// TIA Portal V17 export
// export: Created 2025-06-26T06:49:17.7875276Z, ExportSetting WithDefaults, DisplayName Totally Integrated Automation Portal, DisplayVersion V17 Update 8, DisplayName TIA Portal Openness, DisplayVersion V17 Update 8, DisplayName TIA Portal Version Control Interface, DisplayVersion V17, DisplayName STEP 7 Professional, DisplayVersion V17 Update 8, DisplayName STEP 7 Safety, DisplayVersion V17 Update 6, DisplayName WinCC Advanced, DisplayVersion V17 Update 8
FUNCTION "CompressorCalculations" : Void   // FC25, FBD
{ S7_Optimized_Access := 'TRUE' }
VERSION : 0.1
// stored: AutoNumber true, IsIECCheckEnabled false, SetENOAutomatically false, UDAEnableTagReadback false
   VAR_TEMP
      CrankcaseSaturationTemperature : Real;
      SaturationTemperatureSuction : Real;
      SaturationTemperatureDischarge : Real;
      Massflow : Real;
      VolumetricEfficiency : Real;
      HeatRateCompressor : Real;
      IsentropicEfficiencyCompressor : Real;
      FMEP : Real;
   END_VAR
   VAR_TEMP   // added for the SCL form of the ladder/FBD networks
      _w1 : Bool;
   END_VAR
BEGIN

REGION Network 1: Crankcase saturation temperature
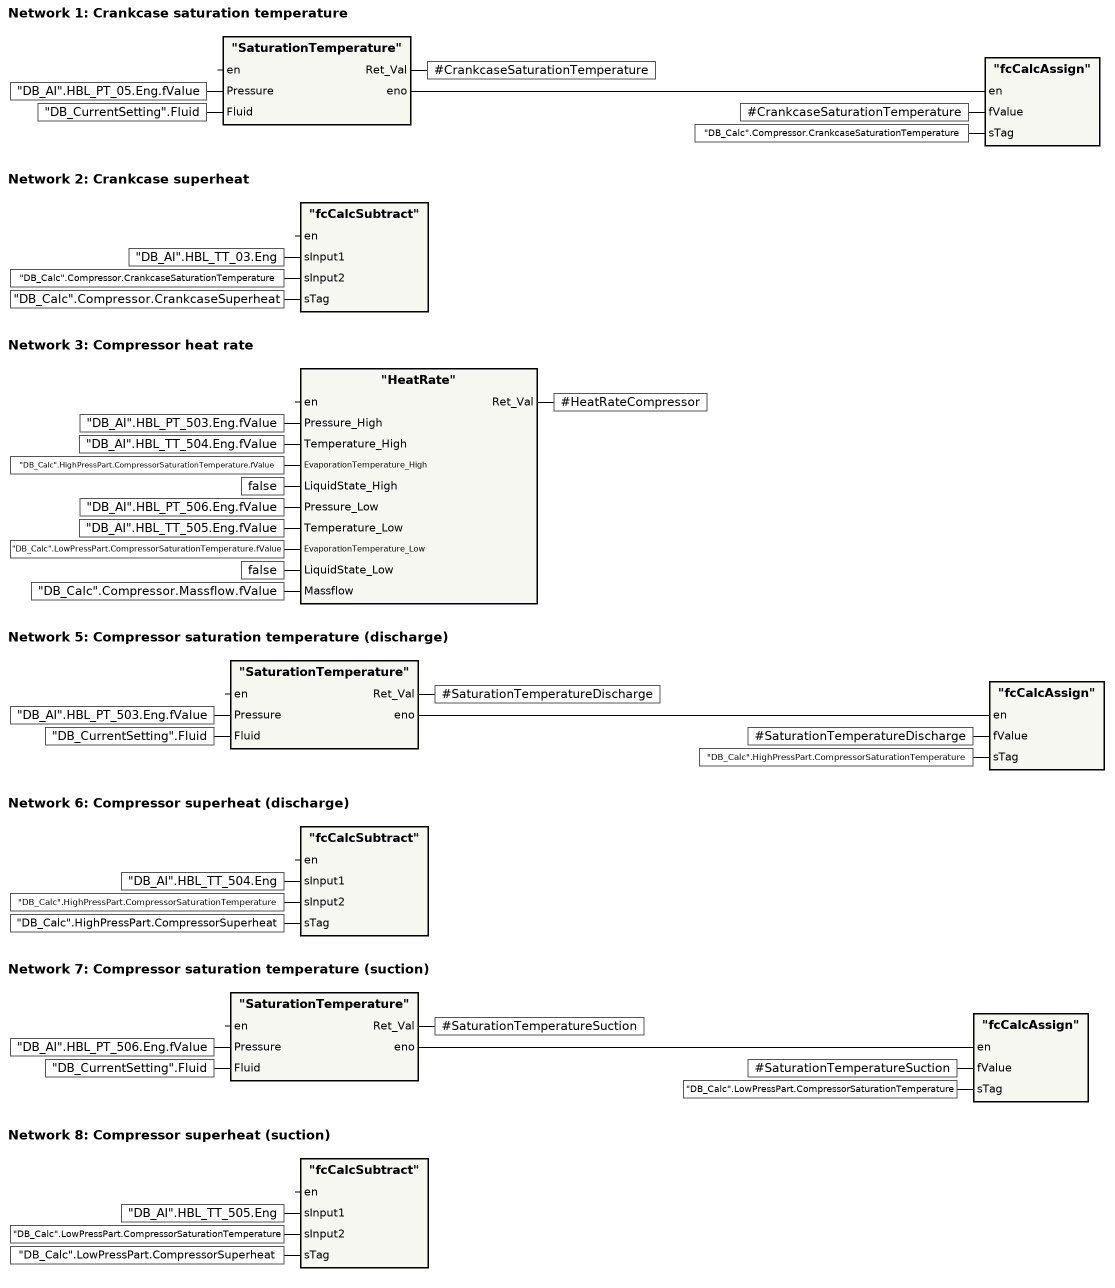
   #CrankcaseSaturationTemperature := "SaturationTemperature"(Pressure := "DB_AI".HBL_PT_05.Eng.fValue,
                           Fluid := "DB_CurrentSetting".Fluid,
                           ENO => #_w1);
   IF #_w1 THEN
       "fcCalcAssign"(fValue := #CrankcaseSaturationTemperature,
                      sTag := "DB_Calc".Compressor.CrankcaseSaturationTemperature);
   END_IF;
END_REGION

REGION Network 2: Crankcase superheat
   // Crankcase temperature is taken to be the same as the oil sump oil temperature
   "fcCalcSubtract"(sInput1 := "DB_AI".HBL_TT_03.Eng,
                    sInput2 := "DB_Calc".Compressor.CrankcaseSaturationTemperature,
                    sTag := "DB_Calc".Compressor.CrankcaseSuperheat);
END_REGION

REGION Network 3: Compressor heat rate
   // The high side is the compressor discharge temp & pressure, gas phase
   // The low side is the compressor suction temp & pressure, gas phase
   #HeatRateCompressor := "HeatRate"(Pressure_High := "DB_AI".HBL_PT_503.Eng.fValue,
                           Temperature_High := "DB_AI".HBL_TT_504.Eng.fValue,
                           EvaporationTemperature_High := "DB_Calc".HighPressPart.CompressorSaturationTemperature.fValue,
                           LiquidState_High := false,
                           Pressure_Low := "DB_AI".HBL_PT_506.Eng.fValue,
                           Temperature_Low := "DB_AI".HBL_TT_505.Eng.fValue,
                           EvaporationTemperature_Low := "DB_Calc".LowPressPart.CompressorSaturationTemperature.fValue,
                           LiquidState_Low := false,
                           Massflow := "DB_Calc".Compressor.Massflow.fValue);
END_REGION

REGION Network 4 (SCL): Isentropic efficiency
   IF "DB_Calc".System.ElectricalPower.fValue > 0.0 THEN
       #IsentropicEfficiencyCompressor := #HeatRateCompressor / "DB_Calc".System.ElectricalPower.fValue * 100.0;
   ELSE
       #IsentropicEfficiencyCompressor := 0.0;
   END_IF;

   "fcCalcAssign"(fValue := #IsentropicEfficiencyCompressor, sTag := "DB_Calc".Compressor.IsentropicEfficiency);
END_REGION

REGION Network 5: Compressor saturation temperature (discharge)
   // High press part
   #SaturationTemperatureDischarge := "SaturationTemperature"(Pressure := "DB_AI".HBL_PT_503.Eng.fValue,
                           Fluid := "DB_CurrentSetting".Fluid,
                           ENO => #_w1);
   IF #_w1 THEN
       "fcCalcAssign"(fValue := #SaturationTemperatureDischarge,
                      sTag := "DB_Calc".HighPressPart.CompressorSaturationTemperature);
   END_IF;
END_REGION

REGION Network 6: Compressor superheat (discharge)
   // Superheat out = Compressor discharge temperature - compressor saturation temperature
   "fcCalcSubtract"(sInput1 := "DB_AI".HBL_TT_504.Eng,
                    sInput2 := "DB_Calc".HighPressPart.CompressorSaturationTemperature,
                    sTag := "DB_Calc".HighPressPart.CompressorSuperheat);
END_REGION

REGION Network 7: Compressor saturation temperature (suction)
   #SaturationTemperatureSuction := "SaturationTemperature"(Pressure := "DB_AI".HBL_PT_506.Eng.fValue,
                           Fluid := "DB_CurrentSetting".Fluid,
                           ENO => #_w1);
   IF #_w1 THEN
       "fcCalcAssign"(fValue := #SaturationTemperatureSuction,
                      sTag := "DB_Calc".LowPressPart.CompressorSaturationTemperature);
   END_IF;
END_REGION

REGION Network 8: Compressor superheat (suction)
   // Superheat in = Compressor suction temperature - compressor saturation temperature
   "fcCalcSubtract"(sInput1 := "DB_AI".HBL_TT_505.Eng,
                    sInput2 := "DB_Calc".LowPressPart.CompressorSaturationTemperature,
                    sTag := "DB_Calc".LowPressPart.CompressorSuperheat);
END_REGION

REGION Network 9: Massflow & volumetric efficiency
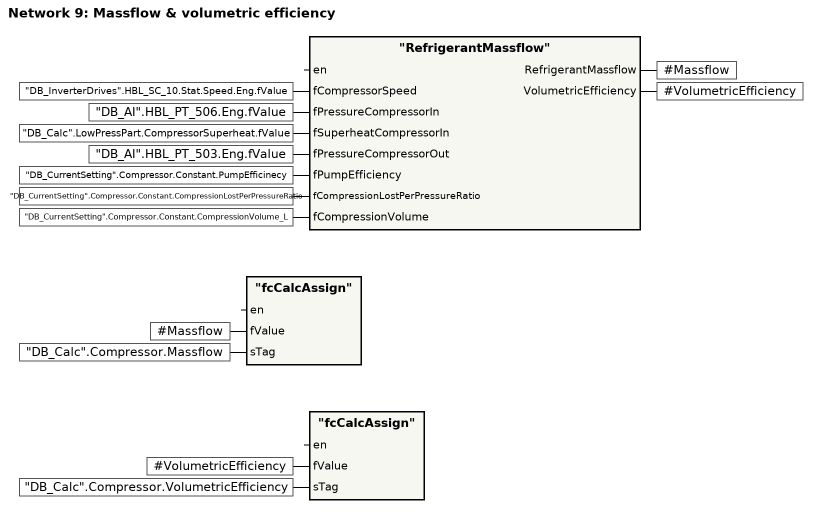
   "RefrigerantMassflow"(fCompressorSpeed := "DB_InverterDrives".HBL_SC_10.Stat.Speed.Eng.fValue,
                         fPressureCompressorIn := "DB_AI".HBL_PT_506.Eng.fValue,
                         fSuperheatCompressorIn := "DB_Calc".LowPressPart.CompressorSuperheat.fValue,
                         fPressureCompressorOut := "DB_AI".HBL_PT_503.Eng.fValue,
                         fPumpEfficiency := "DB_CurrentSetting".Compressor.Constant.PumpEfficinecy,
                         fCompressionLostPerPressureRatio := "DB_CurrentSetting".Compressor.Constant.CompressionLostPerPressureRatio,
                         fCompressionVolume := "DB_CurrentSetting".Compressor.Constant.CompressionVolume_L,
                         RefrigerantMassflow => #Massflow,
                         VolumetricEfficiency => #VolumetricEfficiency);
   "fcCalcAssign"(fValue := #Massflow, sTag := "DB_Calc".Compressor.Massflow);
   "fcCalcAssign"(fValue := #VolumetricEfficiency, sTag := "DB_Calc".Compressor.VolumetricEfficiency);
END_REGION

REGION Network 10 (SCL): FMEP
   // IMEP is estimated as follows:
   // IMEP ~(discharge pressure + suction pressure)/2
   // BMEP = Torque * 0.37793 kPa/Nm
   // FMEP = IMEP - BMEP
   // FMEP = (discharge pressure + suction pressure)/2 - Torque * 0.37793 kPa/Nm

   #FMEP := ("DB_AI".HBL_PT_506.Eng.fValue + "DB_AI".HBL_PT_503.Eng.fValue)/2 - "DB_InverterDrives".HBL_SC_10.Stat.Torque.Eng.fValue/100 * 3407 * 0.37793;
   "fcCalcAssign"(fValue := #FMEP, sTag := "DB_Calc".System.FMEP);
END_REGION
END_FUNCTION
